TYPE "PPrf_A0301_0302_Assemblaggio"
VERSION : 0.1
// Block: PPrf_A0301_0302_Assemblaggio
   STRUCT
      Trasporto : PPrf_A0301_Trasporto;
      Ribaltatore : PPrf_A0301_Ribaltatore;
      Bordatrice : PPrf_A0302_Bordatrice;
      HU_Cytropack : Struct
         Target_PressureParegg : Real;
         Target_MaxSpeedLimit : Real;
      END_STRUCT;
   END_STRUCT;

END_TYPE
